Universal Robots PolyScope program: socket_test.urp

Program socket_test (installation=default directory=/programs createdIn=5.2.1.61344 lastSavedIn=5.2.1.61344 robotSerialNumber=20185500910)
Calibrated DH parameters: a=[0.000049, -0.2988, -0.136614, -0.000051, 0.000155, 0]; d=[0.162579, 88.949821, -241.716128, 152.899954, 0.099639, 0.099482]; alpha=[1.56987, -0.003405, -0.002407, 1.569674, -1.569166, 0]; deltaTheta=[0, -0.792152, 8.290367, -1.215029, 0.000002, 0]
BeforeStart
  var_1 := socket_open("192.168.56.1",30000)
Robot Program (runOnlyOnce=false)
  Loop While (checkContinuously=false) expression=(var_1≟ False )
    var_1 := socket_open("192.168.56.1",30000)
    Wait Sleep waitTime=0.5
  pose1 := get_actual_tcp_pose()
  joints1 := get_actual_joint_positions()
  Script: socket_send_string(pose1)
  Wait Sleep waitTime=0.5
  Script: socket_send_string(joints1)
  Wait Sleep waitTime=0.5
  Script: socket_send_string("asking_for_data")
  Wait Sleep waitTime=0.5
  var_2 := socket_read_ascii_float(3)
  Wait Sleep waitTime=0.5
  var_1 := False
  Script: socket_close()
